{region '#Template'}
	{attribute 'Version' := '5.0.0.0'}
	{attribute 'Tags' := '"LCID": "1031", "Text": "Trade, Plant, AC"'}
	{attribute 'Tags' := '"LCID": "1033", "Text": "Trade, Plant, AC"'}
	{attribute 'Using' := '"Type": "Template", "URI": "Site"'}
	{attribute 'Description' := '"LCID": "1031", "Text": "Aufruf der Anlagen des Gewerks Klimaanlagen"'}
	{attribute 'Description' := '"LCID": "1033", "Text": "Calling the plants of the trade air conditioning"'}
{endregion}
FUNCTION_BLOCK FB_BA_AirConditioning EXTENDS FB_BA_View
VAR_INPUT CONSTANT
	AHU01				: FB_BA_AHU_1st_10;
END_VAR
VAR_INPUT
END_VAR
VAR_OUTPUT
END_VAR
VAR
END_VAR

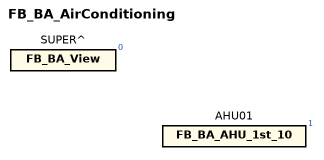
SUPER^(); // FB_BA_View
AHU01(); // FB_BA_AHU_1st_10

METHOD FB_init : BOOL
VAR_INPUT
	bInitRetains : BOOL; // if TRUE, the retain variables are initialized (warm start / cold start)
	bInCopyCode : BOOL;  // if TRUE, the instance afterwards gets moved into the copy code (online change)
END_VAR
AHU01.iParent 					:= THIS^;	                               
AHU01.iLabel					:= LblPlt_Partial_air_conditioning_system;	
AHU01.sObjectName				:= '{Idx=01}';                       
AHU01.eDPADMode					:= E_BA_DPADMode.eInclude;
END_METHOD

END_FUNCTION_BLOCK

(* stored: Version 1.1.0.1, ProductVersion 3.1.4024.12
   POU FB_BA_AirConditioning: Id {bdc7bc27-4147-48f1-9968-568ce857494b}, SpecialFunc None
   Method FB_init: Id {0439e4e3-25f8-4f0e-a8ed-d1c0ce404fd0} *)
